{attribute 'qualified_only'}
//{attribute 'strict'}
{attribute 'to_string'}
TYPE A21 :
(
	IDLE,
	STAGE_BUNK,
	REMOVE_BUNK_FROM_STAGE,
	
	LOAD_BUNK_TO_TOP := 4,
	LOAD_BUNK_TO_SIDE,
	LOAD_BUNK_TO_BOTTOM,
	REMOVE_BUNK_FROM_TOP,
	REMOVE_BUNK_FROM_SIDE,
	REMOVE_BUNK_FROM_BOTTOM,
	
	GET_CHIPBOARD_FROM_SKID := 11,
	REMOVE_CHIPBOARD_FROM_TOOL,
	PLACE_CHIPBOARD_TO_TOP,
	PLACE_CHIPBOARD_TO_BOTTOM,
	REMOVE_CHIPBOARD_TOP,
	REMOVE_CHIPBOARD_BOTTOM,
	
	FIX_CHIPBOARD_ORIENTATION := 19,
	
	//testing only
	MOVE_HOME := 21,
	MOVE_POSITION1,
	MOVE_POSITION2,
	MOVE_UP,
	MOVE_DOWN,
	
	DIRECT_BUNK_TO_TOP := 27,
	DIRECT_BUNK_TO_SIDE,
	DIRECT_BUNK_TO_BOTTOM,
	
	INSPECT_BUNK := 31,
	INSPECT_CHIPBOARD,
	
	TOOL_CHANGE_BUNK := 34,
	TOOL_CHANGE_CHIPBOARD,
	
	size
);
END_TYPE

(* stored: Version 1.1.0.1, ProductVersion 3.1.4024.11
   DUT A21: Id {3aef6316-63c5-464d-a387-89abc0a97ce4} *)
